(* IEC 61131-3 sources: com.logicals.lc3.webinar/usRTS_RPMControl_iSOC/src_FB_LIB_SAFE/Numeric/LREAL, 8 files *)

(* ---- wADD_LREAL_2.iecst ---- *)
NAMESPACE logicals.web.standard
NAMESPACE numeric

/*
 * Function block wrapper for IEC 61131-3 ADD<br>
 * IN1 =  1st value (LREAL)<br>
 * IN2 =  2nd value (LREAL)<br>
 * OUT = Sum of all input values (LREAL)<br>
 */
FUNCTION_BLOCK wADD_LREAL_2
	{ vNameAlignment:="center"; altName:="+"; bgColor:="Orange"; width:=40; hideIONames; }
	VAR_INPUT
		IN1 : LREAL;
		IN2 : LREAL;
	END_VAR
	VAR_OUTPUT
		OUT : LREAL;
	END_VAR

	OUT := ADD(IN1:=IN1, IN2:=IN2, ENO=>ENO);
END_FUNCTION_BLOCK

END_NAMESPACE
END_NAMESPACE

(* ---- wADD_LREAL_3.iecst ---- *)
NAMESPACE logicals.web.standard
NAMESPACE numeric

/*
 * Function block wrapper for IEC 61131-3 ADD<br>
 * IN1 =  1st value (LREAL)<br>
 * IN2 =  2nd value (LREAL)<br>
 * IN3 =  3rd value (LREAL)<br>
 * OUT = Sum of all input values (LREAL)<br>
 */
FUNCTION_BLOCK wADD_LREAL_3
	{ vNameAlignment:="center"; altName:="+"; bgColor:="Orange"; width:=40; hideIONames; }
	VAR_INPUT
		IN1 : LREAL;
		IN2 : LREAL;
		IN3 : LREAL;
	END_VAR
	VAR_OUTPUT
		OUT : LREAL;
	END_VAR

	OUT := ADD(IN1:=IN1, IN2:=IN2, IN3:=IN3, ENO=>ENO);
END_FUNCTION_BLOCK

END_NAMESPACE
END_NAMESPACE

(* ---- wADD_LREAL_4.iecst ---- *)
NAMESPACE logicals.web.standard
NAMESPACE numeric

/*
 * Function block wrapper for IEC 61131-3 ADD<br>
 * IN1 =  1st value (LREAL)<br>
 * IN2 =  2nd value (LREAL)<br>
 * IN3 =  3rd value (LREAL)<br>
 * IN4 =  4th value (LREAL)<br>
 * OUT = Sum of all input values (LREAL)<br>
 */
FUNCTION_BLOCK wADD_LREAL_4
	{ vNameAlignment:="center"; altName:="+"; bgColor:="Orange"; width:=40; hideIONames; }
	VAR_INPUT
		IN1 : LREAL;
		IN2 : LREAL;
		IN3 : LREAL;
		IN4 : LREAL;
	END_VAR
	VAR_OUTPUT
		OUT : LREAL;
	END_VAR

	OUT := ADD(IN1:=IN1, IN2:=IN2, IN3:=IN3, IN4:=IN4, ENO=>ENO);
END_FUNCTION_BLOCK

END_NAMESPACE
END_NAMESPACE

(* ---- wDIV_LREAL.iecst ---- *)
NAMESPACE logicals.web.standard
NAMESPACE numeric

/*
 * Function block wrapper for IEC 61131-3 DIV<br>
 * IN1 =  1st value (LREAL)<br>
 * IN2 =  2nd value (LREAL)<br>
 * OUT = quotient of IN1 divided by IN2 (LREAL)<br>
 */
FUNCTION_BLOCK wDIV_LREAL
	{ vNameAlignment:="center"; altName:="/"; bgColor:="Orange"; width:=40; hideIONames; }
	VAR_INPUT
		IN1 : LREAL;
		IN2 : LREAL;
	END_VAR
	VAR_OUTPUT
		OUT : LREAL;
	END_VAR

	OUT := DIV(IN1:=IN1, IN2:=IN2, ENO=>ENO);
END_FUNCTION_BLOCK

END_NAMESPACE
END_NAMESPACE

(* ---- wMUL_LREAL_2.iecst ---- *)
NAMESPACE logicals.web.standard
NAMESPACE numeric

/*
 * Function block wrapper for IEC 61131-3 MUL<br>
 * IN1 =  1st value (LREAL)<br>
 * IN2 =  2nd value (LREAL)<br>
 * OUT = Product of multiplication of all inputs (LREAL)<br>
 */
FUNCTION_BLOCK wMUL_LREAL_2
	{ vNameAlignment:="center"; altName:="*"; bgColor:="Orange"; width:=40; hideIONames; }
	VAR_INPUT
		IN1 : LREAL;
		IN2 : LREAL;
	END_VAR
	VAR_OUTPUT
		OUT : LREAL;
	END_VAR

	OUT := MUL(IN1:=IN1, IN2:=IN2, ENO=>ENO);
END_FUNCTION_BLOCK

END_NAMESPACE
END_NAMESPACE

(* ---- wMUL_LREAL_3.iecst ---- *)
NAMESPACE logicals.web.standard
NAMESPACE numeric

/*
 * Function block wrapper for IEC 61131-3 MUL<br>
 * IN1 =  1st value (LREAL)<br>
 * IN2 =  2nd value (LREAL)<br>
 * IN3 =  3rd value (LREAL)<br>
 * OUT = Product of multiplication of all inputs (LREAL)<br>
 */
FUNCTION_BLOCK wMUL_LREAL_3
	{ vNameAlignment:="center"; altName:="*"; bgColor:="Orange"; width:=40; hideIONames; }
	VAR_INPUT
		IN1 : LREAL;
		IN2 : LREAL;
		IN3 : LREAL;
	END_VAR
	VAR_OUTPUT
		OUT : LREAL;
	END_VAR

	OUT := MUL(IN1:=IN1, IN2:=IN2, IN3:=IN3, ENO=>ENO);
END_FUNCTION_BLOCK

END_NAMESPACE
END_NAMESPACE

(* ---- wMUL_LREAL_4.iecst ---- *)
NAMESPACE logicals.web.standard
NAMESPACE numeric

/*
 * Function block wrapper for IEC 61131-3 MUL<br>
 * IN1 =  1st value (LREAL)<br>
 * IN2 =  2nd value (LREAL)<br>
 * IN3 =  3rd value (LREAL)<br>
 * IN4 =  4th value (LREAL)<br>
 * OUT = Product of multiplication of all inputs (LREAL)<br>
 */
FUNCTION_BLOCK wMUL_LREAL_4
	{ vNameAlignment:="center"; altName:="*"; bgColor:="Orange"; width:=40; hideIONames; }
	VAR_INPUT
		IN1 : LREAL;
		IN2 : LREAL;
		IN3 : LREAL;
		IN4 : LREAL;
	END_VAR
	VAR_OUTPUT
		OUT : LREAL;
	END_VAR

	OUT := MUL(IN1:=IN1, IN2:=IN2, IN3:=IN3, IN4:=IN4, ENO=>ENO);
END_FUNCTION_BLOCK

END_NAMESPACE
END_NAMESPACE

(* ---- wSUB_LREAL.iecst ---- *)
NAMESPACE logicals.web.standard
NAMESPACE numeric

/*
 * Function block wrapper for IEC 61131-3 SUB<br>
 * IN1 =  1st value (LREAL)<br>
 * IN2 =  2nd value (LREAL)<br>
 * OUT = IN1 minus IN2 (LREAL)<br>
 */
FUNCTION_BLOCK wSUB_LREAL
	{ vNameAlignment:="center"; altName:="-"; bgColor:="Orange"; width:=40; hideIONames; }
	VAR_INPUT
		IN1 : LREAL;
		IN2 : LREAL;
	END_VAR
	VAR_OUTPUT
		OUT : LREAL;
	END_VAR

	OUT := SUB(IN1:=IN1, IN2:=IN2, ENO=>ENO);
END_FUNCTION_BLOCK

END_NAMESPACE
END_NAMESPACE
